TYPE ST_MV_MAFAC_GT_Parameter :
STRUCT
	Temp_Kaltwasser        : REAL;
	Temp_Kaltwasser_Max    : REAL;
	Temp_Kaltwasser_Min    : REAL;

END_STRUCT
END_TYPE

(* stored: Version 1.1.0.1, ProductVersion 3.1.4024.9
   DUT ST_MV_MAFAC_GT_Parameter: Id {1299be19-bcff-4b5a-b4dd-32f6e05823f8} *)
